# EPICS substitutions: RadiationMonitoringApp/Db/common/mfht-station.substitutions
file radm_info.template
{
    pattern
    { P,               , LOC     ,TYPE}
    { RADM:SITE:$(UNIT), "Site"  , 5  }
}

file fht6020-system-status.template
{
     pattern { P,                  PORT,      ADDRESS    }
             { RADM:SITE:$(UNIT),  $(FPORT),  01         }
}

file fht6020-channel-status.template
{
      pattern { P,                  PORT,      ADDRESS,   CHANNEL    }
              { RADM:SITE:$(UNIT),  $(FPORT),  01,        01         }
              { RADM:SITE:$(UNIT),  $(FPORT),  01,        02         }
}

file mfht_stat.template
{
      pattern { STATION     }
              { $(UNIT) }
}
